(*
Will be an abstract class that will be used to configure all parts of the machine through json
*)

FUNCTION_BLOCK ABSTRACT FB_ConfigBase
VAR_INPUT
END_VAR
VAR_OUTPUT
END_VAR
VAR 
	_fbName : STRING; //name of FB set on init
END_VAR

METHOD _F_Axis : HRESULT
VAR_IN_OUT
	a_pstAxisParameterSet : POINTER TO Tc2_MC2.ST_AxisParameterSet; //pointer to array
	pstAxisMapping : UDINT;
END_VAR
END_METHOD

METHOD PROTECTED ABSTRACT _F_IO : HResult
VAR_IN_OUT
	a_pstIOMappingJson : POINTER TO ST_IOMappingJson; //pointer to array
	ustIOMappingJson : UDINT; 		
END_VAR
END_METHOD

(*
return the list of vars that want to be saved and loaded 
*)

METHOD PROTECTED ABSTRACT _F_Recipe : HResult
VAR_IN_OUT
	a_pstAnyTypeUser : POINTER TO MPM_JsonParser.ST_AnyType_User; //pointer to array
	uAnyTypeUser : UDINT; //size of array	
END_VAR
VAR_OUTPUT

END_VAR
END_METHOD

METHOD PROTECTED ABSTRACT _F_System : HResult
VAR_IN_OUT
	a_pstAnyTypeUser : POINTER TO MPM_JsonParser.ST_AnyType_User; //pointer to array
	uAnyTypeUser : UDINT; //size of array	
END_VAR
END_METHOD

METHOD PUBLIC FINAL F_AXIS : HRESULT
VAR_INPUT
	lastResult : HRESULT;
	sJson : SJsonValue;
	pfbJsonSchema : POINTER TO FB_NCAxisJson_V2;	
	bGet : BOOL;
END_VAR

VAR_INST
	_fbResult : FB_ResultHelper_V2;
	pResult : POINTER TO HRESULT;
END_VAR

VAR
	a_pstAxisParameterSet : POINTER TO Tc2_MC2.ST_AxisParameterSet;
	dstAxisParameterSet : UDINT; //number of bytes in a_stAnyUser
	
	uSizeOfArray : UDINT;
	
	pstAxisParameterSet : POINTER TO Tc2_MC2.ST_AxisParameterSet; //pointer for loop
	x : UDINT;
END_VAR


VAR CONSTANT
	uSizeOfStAnyType : UDINT := SIZEOF(Tc2_MC2.ST_AxisParameterSet);
END_VAR
IF _fbResult.M_MethodResult(F_AXIS,ADR(pResult),lastResult) = FALSE THEN
	RETURN;
END_IF


pResult^ := _F_Axis(a_pstAxisParameterSet,dstAxisParameterSet);
//pResult^ := MPM_FBResult.E_Result.S_WORKING;
IF bGet = FALSE THEN
	sJson := pfbJsonSchema^.M_SetJsonMember(sJson,_fbName);
	IF a_pstAxisParameterSet > 0 AND dstAxisParameterSet > 0 AND uSizeOfStAnyType > 0 THEN //make sure all values are vaild
		uSizeOfArray := dstAxisParameterSet/uSizeOfStAnyType - 1; //get number of items in array
		FOR x := 0 TO uSizeOfArray BY 1 DO //loop through all items 
			pstAxisParameterSet := a_pstAxisParameterSet + uSizeOfStAnyType*x; // get array position
			pResult^ := pfbJsonSchema^.M_SetAxisJson(pResult^,sJson,pstAxisParameterSet);
		END_FOR
	END_IF	
ELSIF bGet = TRUE THEN
	sJson := pfbJsonSchema^.FindMember(sJson,_fbName);
	IF a_pstAxisParameterSet > 0 AND dstAxisParameterSet > 0 AND uSizeOfStAnyType > 0 THEN //make sure all values are vaild
		uSizeOfArray := dstAxisParameterSet/uSizeOfStAnyType - 1; //get number of items in array
		FOR x := 0 TO uSizeOfArray BY 1 DO //loop through all items 
			pstAxisParameterSet := a_pstAxisParameterSet + uSizeOfStAnyType*x; // get array position
			pResult^ := pfbJsonSchema^.M_GetAxisJson(pResult^,sJson,pstAxisParameterSet);
		END_FOR
	END_IF
END_IF
END_METHOD

METHOD PROTECTED F_Event_ST_AnyType_Compare : HResult
VAR_INPUT
	srcvar : POINTER TO MPM_JsonParser.ST_AnyType_User; //PVOID FOR any value
	desvar : POINTER TO MPM_JsonParser.ST_AnyType_User;	//What was input
END_VAR
VAR
END_VAR
IF srcvar^.typeclass = desvar^.typeclass AND srcvar^.diSize = desvar^.diSize THEN
	desvar^.pvalue := srcvar^.pvalue;
	F_Event_ST_AnyType_Compare := MPM_FBResult.E_Result.S_OK;
ELSE
	F_Event_ST_AnyType_Compare := MPM_FBResult.E_Result.S_FAILED;	
END_IF
END_METHOD

METHOD PUBLIC F_GetArrayLength : HResult
VAR_INPUT
	sizeOfInst : DINT;
	sizeOFType : DINT;
END_VAR
VAR_OUTPUT
	length : DINT;
END_VAR
VAR
	_numOfElements : DINT;
END_VAR
IF sizeOFType > 0 AND sizeOfInst > 0 THEN
	_numOfElements := sizeOfInst/sizeOFType -1;
	IF _numOfElements > 0 THEN
		length := _numOfElements;
		F_GetArrayLength := MPM_FBResult.E_Result.S_OK;
	END_IF
ELSE
	F_GetArrayLength := MPM_FBResult.E_Result.S_FAILED;
	RETURN;
END_IF
END_METHOD

METHOD PUBLIC F_GetArrayPosition : HResult
VAR_INPUT
	sizeOfInst : DINT;
	sizeOFType : DINT;
	index : DINT;
END_VAR
VAR_OUTPUT
	offset : DINT;
	length : DINT;
END_VAR
VAR
END_VAR
F_GetArrayPosition := F_GetArrayLength(sizeOfInst,sizeOFType, length => length);
IF F_GetArrayPosition = MPM_FBResult.E_Result.S_OK THEN
	IF index >= 0 AND index <= length THEN
		offset := sizeOFType*index;
	ELSE
		F_GetArrayPosition := MPM_FBResult.E_Result.S_FAILED;
	END_IF
ELSE
	F_GetArrayPosition := MPM_FBResult.E_Result.S_OK;
END_IF
END_METHOD

METHOD PUBLIC FINAL F_IO : HRESULT
VAR_INPUT
	lastResult : HRESULT;
	sJson : SJsonValue;
	pfbJsonSchema : POINTER TO FB_JsonSchemaEx_OLD;
	bGet : BOOL;	
END_VAR

VAR_INST
	_fbResult : FB_ResultHelper_V2;
	pResult : POINTER TO HRESULT;
END_VAR

VAR
	a_pstIOMappingJson : POINTER TO ST_IOMappingJson; // pointer to array of vars
	uAnyTypeUser : UDINT; //number of bytes in a_stAnyUser
	
	uSizeOfArray : UDINT;
	pstIOMappingJson : POINTER TO ST_IOMappingJson; //pointer for loop
	x : UDINT;
END_VAR


VAR CONSTANT
	uSizeOfStAnyType : UDINT := SIZEOF(ST_IOMappingJson);
END_VAR
IF _fbResult.M_MethodResult(F_IO,ADR(pResult),lastResult) = FALSE THEN
	RETURN;
END_IF


pResult^ := _F_IO(a_pstIOMappingJson,uAnyTypeUser); //gets pointer from FB


pResult^ := MPM_FBResult.E_Result.S_WORKING;
//set
IF bGet = FALSE THEN
	sJson := pfbJsonSchema^.M_SetJsonMember(sJson,_fbName);
	IF a_pstIOMappingJson > 0 AND_THEN uAnyTypeUser > 0 AND uSizeOfStAnyType > 0 THEN //make sure all values are vaild
		uSizeOfArray := uAnyTypeUser/uSizeOfStAnyType - 1; //get number of items in array
		FOR x := 0 TO uSizeOfArray BY 1 DO //loop through all items 
			pstIOMappingJson := a_pstIOMappingJson + uSizeOfStAnyType*x; // get array position
			sJson := pfbJsonSchema^.M_SetJsonMember(sJson,pstIOMappingJson^.name); //set json value
			pfbJsonSchema^.M_SetJsonMemberValue(sJson,'channel',pstIOMappingJson^.channel); //set json value
			pfbJsonSchema^.M_SetJsonMemberValue(sJson,'deviceNum',pstIOMappingJson^.deviceNum); //set json value
			pfbJsonSchema^.M_SetJsonMemberValue(sJson,'ethercatDeviceNum',pstIOMappingJson^.ethercatDeviceNum); //set json value
			pfbJsonSchema^.M_SetJsonMemberValue(sJson,'ioLinkDevice',pstIOMappingJson^.ioLinkDevice); //set json value
			pfbJsonSchema^.M_SetJsonMemberValue(sJson,'ioLinkSlaveChannel',pstIOMappingJson^.ioLinkSlaveChannel); //set json value
		END_FOR
		pResult^ := MPM_FBResult.E_Result.S_OK;
	ELSE
		pResult^ := MPM_FBResult.E_Result.S_FAILED;
	END_IF
//get
ELSIF bGet = TRUE THEN
	sJson := pfbJsonSchema^.FindMember(sJson,_fbName);
	IF a_pstIOMappingJson > 0 AND_THEN uAnyTypeUser > 0 AND uSizeOfStAnyType > 0 THEN //make sure all values are vaild
		uSizeOfArray := uAnyTypeUser/uSizeOfStAnyType - 1; //get number of items in array
		FOR x := 0 TO uSizeOfArray BY 1 DO //loop through all items 
			pstIOMappingJson := a_pstIOMappingJson + uSizeOfStAnyType*x; // get array position
			sJson := pfbJsonSchema^.M_SetJsonMember(sJson,pstIOMappingJson^.name); //set json value
			pfbJsonSchema^.M_GetJsonMemberValue(sJson,'channel',pstIOMappingJson^.channel); //set json value
			pfbJsonSchema^.M_GetJsonMemberValue(sJson,'deviceNum',pstIOMappingJson^.deviceNum); //set json value
			pfbJsonSchema^.M_GetJsonMemberValue(sJson,'ethercatDeviceNum',pstIOMappingJson^.ethercatDeviceNum); //set json value
			pfbJsonSchema^.M_GetJsonMemberValue(sJson,'ioLinkDevice',pstIOMappingJson^.ioLinkDevice); //set json value
			pfbJsonSchema^.M_GetJsonMemberValue(sJson,'ioLinkSlaveChannel',pstIOMappingJson^.ioLinkSlaveChannel); //set json value
		END_FOR
		pResult^ := MPM_FBResult.E_Result.S_OK;
	ELSE
		pResult^ := MPM_FBResult.E_Result.S_FAILED;
	END_IF
END_IF
END_METHOD

METHOD PROTECTED F_Map_ST_IOMappingJson : HRESULT
VAR_INPUT
	stIOMappingJson : POINTER TO ST_IOMappingJson;
	name : STRING;
	pPVoid : POINTER TO PVOID;
END_VAR
END_METHOD

METHOD PUBLIC FINAL F_Recipe : HRESULT
VAR_INPUT
	lastResult : HRESULT;
	sJson : SJsonValue;
	pfbJsonSchema : POINTER TO FB_JsonSchemaEx_OLD;	
	bGet : BOOL;
END_VAR

VAR_INST
	_fbResult : FB_ResultHelper_V2;
	pResult : POINTER TO HRESULT;
END_VAR

VAR
	a_stAnyUser : POINTER TO MPM_JsonParser.ST_AnyType_User; // pointer to array of vars
	uAnyTypeUser : UDINT; //number of bytes in a_stAnyUser
	
	uSizeOfArray : UDINT;
	pstAnyUser : POINTER TO MPM_JsonParser.ST_AnyType_User; //pointer for loop
	x : UDINT;
END_VAR

VAR CONSTANT
	uSizeOfStAnyType : UDINT := SIZEOF(MPM_JsonParser.ST_AnyType_User);
END_VAR
IF _fbResult.M_MethodResult(F_Recipe,ADR(pResult),lastResult) = FALSE THEN
	RETURN;
END_IF


pResult^ := _F_Recipe(a_stAnyUser,uAnyTypeUser);


pResult^ := MPM_FBResult.E_Result.S_WORKING;

//set
IF bGet = FALSE THEN
	sJson := pfbJsonSchema^.M_SetJsonMember(sJson,_fbName);
	IF a_stAnyUser > 0 AND_THEN uAnyTypeUser > 0 AND uSizeOfStAnyType > 0 THEN //make sure all values are vaild
		uSizeOfArray := uAnyTypeUser/uSizeOfStAnyType - 1; //get number of items in array
		FOR x := 0 TO uSizeOfArray BY 1 DO //loop through all items 
			pstAnyUser := a_stAnyUser + uSizeOfStAnyType*x; // get array position
				pfbJsonSchema^.M_SetJsonMemberValue_AnyType(sJson,pstAnyUser^.name,pstAnyUser^); //set json value
		END_FOR
		pResult^ := MPM_FBResult.E_Result.S_OK;
	ELSE
		pResult^ := MPM_FBResult.E_Result.S_FAILED;
	END_IF
	
//get
ELSIF bGet = TRUE THEN 	
	sJson := pfbJsonSchema^.FindMember(sJson,_fbName);
	IF a_stAnyUser > 0 AND_THEN uAnyTypeUser > 0 AND uSizeOfStAnyType > 0 THEN //make sure all values are vaild
		uSizeOfArray := uAnyTypeUser/uSizeOfStAnyType - 1; //get number of items in array
		FOR x := 0 TO uSizeOfArray BY 1 DO //loop through all items 
			pstAnyUser := a_stAnyUser + uSizeOfStAnyType*x; // get array position
				pfbJsonSchema^.M_GetJsonMemberValue_AnyType(sJson,pstAnyUser^.name,pstAnyUser^); //set json value
		END_FOR
		pResult^ := MPM_FBResult.E_Result.S_OK;
	ELSE
		pResult^ := MPM_FBResult.E_Result.S_FAILED;
	END_IF
END_IF
END_METHOD

METHOD PUBLIC FINAL F_System : HRESULT
VAR_INPUT
	lastResult : HRESULT;
	sJson : SJsonValue;
	pfbJsonSchema : POINTER TO FB_JsonSchemaEx_OLD;	
	bGet : BOOL;	
END_VAR

VAR_INST
	_fbResult : FB_ResultHelper_V2;
	pResult : POINTER TO HRESULT;
END_VAR

VAR
	a_stAnyUser : POINTER TO MPM_JsonParser.ST_AnyType_User; // pointer to array of vars
	uAnyTypeUser : UDINT; //number of bytes in a_stAnyUser
	
	uSizeOfArray : UDINT;
	pstAnyUser : POINTER TO MPM_JsonParser.ST_AnyType_User; //pointer for loop
	x : UDINT;
END_VAR


VAR CONSTANT
	uSizeOfStAnyType : UDINT := SIZEOF(MPM_JsonParser.ST_AnyType_User);
END_VAR
IF _fbResult.M_MethodResult(F_System,ADR(pResult),lastResult) = FALSE THEN
	RETURN;
END_IF


pResult^ := _F_System(a_stAnyUser,uAnyTypeUser);
//set
IF bGet = FALSE THEN
	pResult^ := MPM_FBResult.E_Result.S_WORKING;
	sJson := pfbJsonSchema^.M_SetJsonMember(sJson,_fbName);
	IF a_stAnyUser > 0 AND_THEN uAnyTypeUser > 0 AND uSizeOfStAnyType > 0 THEN //make sure all values are vaild
		uSizeOfArray := uAnyTypeUser/uSizeOfStAnyType - 1; //get number of items in array
		FOR x := 0 TO uSizeOfArray BY 1 DO //loop through all items 
			pstAnyUser := a_stAnyUser + uSizeOfStAnyType*x; // get array position
				pfbJsonSchema^.M_SetJsonMemberValue_AnyType(sJson,pstAnyUser^.name,pstAnyUser^); //set json value
		END_FOR
		pResult^ := MPM_FBResult.E_Result.S_OK;
	ELSE
		pResult^ := MPM_FBResult.E_Result.S_FAILED;
	END_IF

//get	
ELSIF bGet = TRUE THEN
	sJson := pfbJsonSchema^.FindMember(sJson,_fbName);
	IF a_stAnyUser > 0 AND_THEN uAnyTypeUser > 0 AND uSizeOfStAnyType > 0 THEN //make sure all values are vaild
		uSizeOfArray := uAnyTypeUser/uSizeOfStAnyType - 1; //get number of items in array
		FOR x := 0 TO uSizeOfArray BY 1 DO //loop through all items 
			pstAnyUser := a_stAnyUser + uSizeOfStAnyType*x; // get array position
				pfbJsonSchema^.M_GetJsonMemberValue_AnyType(sJson,pstAnyUser^.name,pstAnyUser^); //set json value
		END_FOR
		pResult^ := MPM_FBResult.E_Result.S_OK;
	ELSE
		pResult^ := MPM_FBResult.E_Result.S_FAILED;
	END_IF	
END_IF
END_METHOD

METHOD PROTECTED F_TO_LREAL : LREAL
VAR_INPUT
	pPvoid : PVOID;
END_VAR
VAR_OUTPUT
	error : BOOL;
END_VAR
VAR
	pLREAL : POINTER TO LREAL;
END_VAR
IF pPvoid > 0 THEN
	pLREAL := pPvoid;
	F_TO_LREAL := pLREAL^;
ELSE
	error := TRUE;
END_IF
END_METHOD

METHOD FB_init : BOOL
VAR_INPUT
	bInitRetains : BOOL; // if TRUE, the retain variables are initialized (warm start / cold start)
	bInCopyCode : BOOL;  // if TRUE, the instance afterwards gets moved into the copy code (online change)
	fbName : STRING;
END_VAR
_fbName := fbName;
END_METHOD

METHOD PUBLIC ABSTRACT M_Events : HResult
VAR_INPUT
	lastResult : HResult;
	eventID : DINT;
END_VAR
END_METHOD

METHOD PUBLIC ABSTRACT M_Execute : HRESULT
VAR_INPUT
END_VAR
VAR_INST

END_VAR
END_METHOD

METHOD PUBLIC ABSTRACT M_GetEvent : HResult
VAR_INPUT
	pFbDiscreteEvents : POINTER TO POINTER TO FB_DiscreteEvents;
	index : DINT;	
END_VAR
END_METHOD

PROPERTY PUBLIC P_fbName : STRING
GET
P_fbName := _fbName;
END_GET
END_PROPERTY

PROPERTY PUBLIC ABSTRACT P_GetNumOfEvents : DINT
GET
END_GET
END_PROPERTY

END_FUNCTION_BLOCK

(* stored: Version 1.1.0.1, ProductVersion 3.1.4024.12
   POU FB_ConfigBase: Id {3ccc0d41-27f9-41ab-b33f-1e963a615b44}, SpecialFunc None
   Folder ABSTRACT: Id {d3f0e259-1061-426a-b7a1-3591a9d5be2f}
   Folder Any_Type_Functions: Id {f7907fbb-3c6d-493c-97e3-9d5f2bc80f20}
   Folder Protected: Id {d31bea82-4c8d-4864-8213-7cfbba3c0754}
   Method _F_Axis: Id {7fa39416-568e-4119-8393-652fc6472acb}
   Method _F_IO: Id {25f7451c-b2be-4782-91c3-53451c901d29}
   Method _F_Recipe: Id {acb8c5d6-5487-4d41-9ec0-f4a34dd65731}
   Method _F_System: Id {c67585fa-6db9-4ba3-8b65-2665a130374f}
   Method F_AXIS: Id {c0243cb9-9b32-4370-9384-0993220a2226}
   Method F_Event_ST_AnyType_Compare: Id {d5d96574-3807-41bd-83c3-530358c10783}
   Method F_GetArrayLength: Id {e7ef948f-69e6-4d9b-805d-c192c058829a}
   Method F_GetArrayPosition: Id {1d4567af-9cb4-46e8-a5eb-55d4c46ee846}
   Method F_IO: Id {3a02837e-fabe-4f90-b88e-c4f1e99bdab4}
   Method F_Map_ST_IOMappingJson: Id {5c1ae8e3-b5c1-4247-821a-ef4678ae72df}
   Method F_Recipe: Id {23f9deca-2586-4a9d-b0ee-68078bcc9c57}
   Method F_System: Id {4f92d8d9-026e-4619-8a71-a0cfc6eb2eed}
   Method F_TO_LREAL: Id {5a0750dc-9829-419c-aa77-7ef75aa663e8}
   Method FB_init: Id {39c76da8-be3f-4311-946f-56a7e0460487}
   Method M_Events: Id {9bfb2769-0fba-4d76-86ce-22f9c6c76e6b}
   Method M_Execute: Id {c363a4a8-f039-42db-96a8-a63845351f9a}
   Method M_GetEvent: Id {f2004318-5ed6-456d-af31-fbab4ca91ec4}
   Property P_fbName: Id {5a2b393b-8b77-4ed7-a71a-7e64119bd062}
   Get Get: Id {831f96df-87bd-4bb9-ad06-74017936567e}
   Property P_GetNumOfEvents: Id {5a161ac0-d453-4b8e-913c-bdb5803bb6fd}
   Get Get: Id {4e2a464b-f9ab-44cf-8e2f-328e0d6c78fb} *)
